FUNCTION F_Add1 : DINT
VAR_INPUT
	x : REFERENCE TO DINT;
END_VAR

F_Add1.F_Add1 := x;
x := x + 1;

END_FUNCTION

(* stored: Version 1.1.0.1, ProductVersion 3.1.4024.12
   POU F_Add1: Id {c2100bb4-51ae-4094-aef7-50eb2de6985c}, SpecialFunc None *)
